// TIA Portal V18 export
// export: Created 2026-06-07T16:19:25.8557134Z, ExportSetting WithDefaults, DisplayName Totally Integrated Automation Portal, DisplayVersion V18, DisplayName TIA Portal Openness, DisplayVersion V18, DisplayName TIA Portal Version Control Interface, DisplayVersion V18, DisplayName STEP 7 Professional, DisplayVersion V18, DisplayName STEP 7 Safety, DisplayVersion V18, DisplayName WinCC Professional, DisplayVersion V18
VAR_GLOBAL   // PLC tag table "Default tag table"
   System_Byte AT %MB1 : Byte;
   FirstScan AT %M1.0 : Bool;
   DiagStatusUpdate AT %M1.1 : Bool;
   AlwaysTRUE AT %M1.2 : Bool;
   AlwaysFALSE AT %M1.3 : Bool;
   Clock_Byte AT %MB0 : Byte;
   Clock_10Hz AT %M0.0 : Bool;
   Clock_5Hz AT %M0.1 : Bool;
   "Clock_2.5Hz" AT %M0.2 : Bool;
   Clock_2Hz AT %M0.3 : Bool;
   "Clock_1.25Hz" AT %M0.4 : Bool;
   Clock_1Hz AT %M0.5 : Bool;
   "Clock_0.625Hz" AT %M0.6 : Bool;
   "Clock_0.5Hz" AT %M0.7 : Bool;
   MB_Write_Req AT %M10.0 : Bool;
   MB_Read_Req AT %M10.1 : Bool;
   MB_Write_Done AT %M10.2 : Bool;
   MB_Write_Busy AT %M10.3 : Bool;
   MB_Write_Error AT %M10.4 : Bool;
   MB_Read_Done AT %M10.5 : Bool;
   MB_Read_Busy AT %M10.6 : Bool;
   MB_Read_Error AT %M10.7 : Bool;
   MB_Write_Status AT %MW12 : Word;
   MB_Read_Status AT %MW14 : Word;
END_VAR
